RoboDK station: Examen.rdk

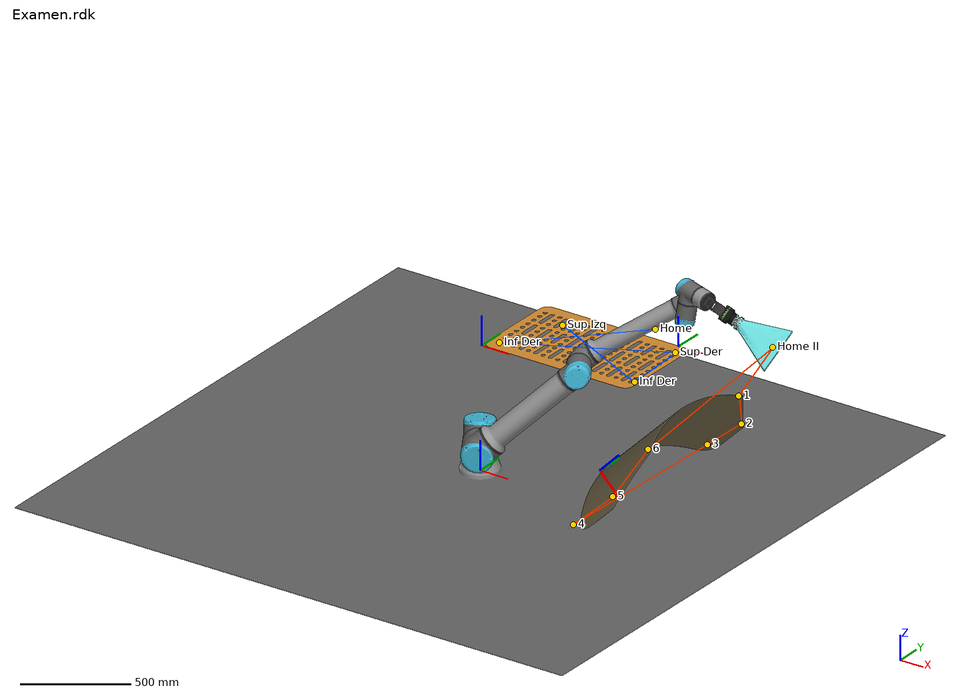
[picture v0: the station drawn from its stored meshes, robots at their saved joint values, targets as dots, program paths as lines]
Station Parcial Juan Pablo Waller (saved by RoboDK 5.7.1). Poses are relative to the parent item; angles as X-Y-Z fixed-axis rotations.
Station parameters (name, value as stored): Palletizing Plugin
  - frame UR10e Base at (0, 0, 0) mm
    - robot UR10e: 6 axes, payload 10 kg, reach 1300 mm, repeatability 0.05 mm, weight 28.9 kg
        modified DH rows (alpha deg, a mm, theta deg, d mm): 0, 0, 0, 180.7; 90, 0, 180, 0; 0, 612.6, 0, 0; 0, 571.335, 0, 174.15; -90, 0, 0, 119.85; 90, 0, 180, 116.55
        joint limits [-360, -360, -360, -360, -360, -360] to [360, 360, 360, 360, 360, 360]; home [0, -90, -90, 0, 90, 0]; saved at [31.361, -137.565, -10.612, -40.337, 45.892, 230.247]
      - tool Camera 2, TCP at (0, -175.95, 321.06) mm, rotated rx 40 ry 0 rz 0 deg, size 215.7 x 276.1 x 372.4 mm
  - frame Frame Inspection A at (-380.72, 555.26, 295.21) mm
    - object Inspection A at (0, 0, 0) mm, size 800 x 500 x 0 mm, geometry from Inspection A.step
    - target Sup Izq (Cartesian target) at (174.15, 387.58, -3.32) mm, rotated rx 130 ry 0 rz 180 deg; joints [130.844, -103.217, -125.462, 48.679, 49.156, 180] of UR10e
    - target Inf Der (Cartesian target) at (784.15, 77.58, 6.68) mm, rotated rx 130 ry 0 rz 180 deg; joints [48.69, -93.865, -135.554, 49.418, 131.31, 180] of UR10e
    - target Sup Der (Cartesian target) at (764.15, 428, 6.68) mm, rotated rx 130 ry 0 rz 180 deg; joints [70.042, -111.81, -111.438, 43.249, 109.958, 180] of UR10e
    - target Inf Der (Cartesian target) at (44.15, 77.58, -3.32) mm, rotated rx 130 ry 0 rz 180 deg; joints [176.472, -89.056, -142.138, 51.193, 3.528, 180] of UR10e
    - target Home (Cartesian target) at (970.87, -22.42, 364.06) mm, rotated rx 150.15 ry 22.69 rz 79.14 deg; joints [236.345, -12.126, -72.564, -42.508, 203.513, 206.373] of UR10e
  - frame Frame Inspection B at (727.24, -100, 245.26) mm, rotated rx 0 ry 45.31 rz 0 deg
    - object Inspection B at (0, 0, 600) mm, rotated rx 180 ry 0 rz 180 deg, size 202.5 x 1023.2 x 500 mm, geometry from Inspection B.step
    - target Home II (Cartesian target) at (10.13, 472.84, 858.92) mm, rotated rx 75.69 ry -40.91 rz 115.81 deg; joints [31.361, -137.565, -10.612, -40.337, 45.892, 230.247] of UR10e
    - target 1 (Cartesian target) at (93.47, 396.26, 589.19) mm, rotated rx 92.78 ry 48.59 rz 72.28 deg; joints [191.46, -4.358, -62.214, -92.572, -89.753, 134.053] of UR10e
    - target 2 (Cartesian target) at (190.18, 550.76, 363.19) mm, rotated rx 114.98 ry -20.73 rz 53.54 deg; joints [210.076, -3.048, -40.342, -84.196, -154.348, 220.55] of UR10e
    - target 3 (Cartesian target) at (170.56, 532.01, 134.8) mm, rotated rx 105.98 ry 23.01 rz 42.65 deg; joints [218.15, 23.894, -71.129, -88.674, -158.09, 170.403] of UR10e
    - target 4 (Cartesian target) at (152.99, -459.76, 96.93) mm, rotated rx 110.55 ry 11.5 rz 73.69 deg; joints [131.099, 29.665, -107.42, -71.943, -57.855, 140.919] of UR10e
    - target 5 (Cartesian target) at (162.47, -457.03, 390.61) mm, rotated rx 110.55 ry 11.5 rz 73.69 deg; joints [141.787, 6.337, -71.821, -86.911, -67.216, 146.744] of UR10e
    - target 6 (Cartesian target) at (82.35, -321.57, 607.52) mm, rotated rx 110.55 ry 11.5 rz 73.69 deg; joints [152.179, -16.608, -41.514, -95.814, -76.495, 151.675] of UR10e
    - target Home II (Cartesian target) at (10.13, 472.84, 858.92) mm, rotated rx 75.69 ry -40.91 rz 115.81 deg; joints [31.361, -137.565, -10.612, -40.337, 45.892, 230.247] of UR10e
  - frame World at (0, 0, 0) mm
    - object Floor at (0, 0, -7) mm, size 3000 x 3000 x 4.2 mm, geometry from Floor.step
  - frame Frame 5 at (0, 1555.26, 0) mm
  - program Prog1 (7 instructions, listed below)
  - program Prog2 (10 instructions, listed below)
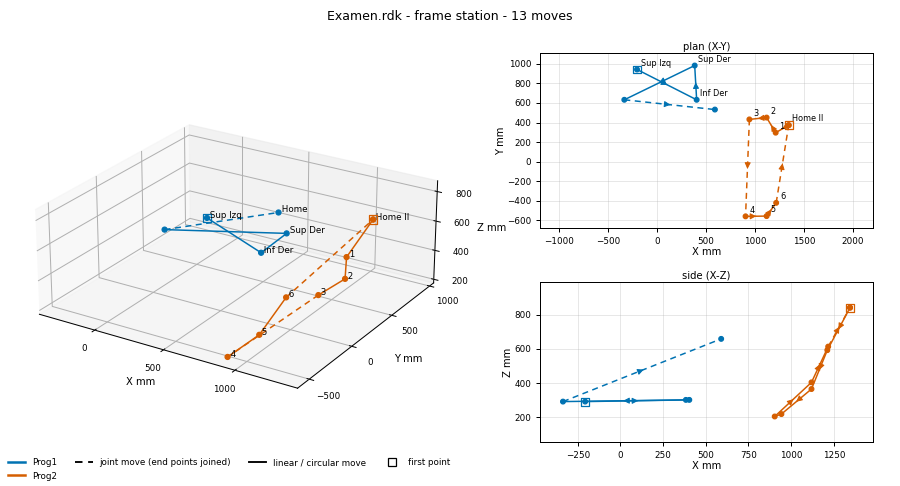
[picture p0: tool path of Examen.rdk in frame station, 13 of 13 moves have a stored position in this frame; points joined in program order, loops and branches not executed]

--- program Prog1 (robot UR10e) ---
  Est. Ref.: Frame Inspection A
  Est. herr: Camera 2
  MoveL (Sup Izq)
  MoveL (Inf Der)
  MoveL (Sup Der)
  MoveL (Inf Der)
  MoveJ (Target 6) -> target Home

--- program Prog2 (robot UR10e) ---
  Est. Ref.: Frame Inspection B
  Est. herr: Camera 2
  MoveJ (Home II)
  MoveL (1)
  MoveL (2)
  MoveL (3)
  MoveJ (4)
  MoveL (5)
  MoveL (6)
  MoveJ (Home II)
